Staubli VAL3: page.pgx

public program page(string& menuname[], num index)
// set all the page in english
begin
  //
  //  PAGE
  //
  //
  // PALLET PAGE
  if index>=10 and index<=19
    title("< Palettenseite >")
  endIf
  // PALLET VIEW PAGE
  if index>=100 and index<=109
    title("< Palettenanzeize >")
  endIf
  switch index
    //
    // PALLET
    //
    // Integrator programmer
    case 10,11
      menuname="Programm anzeigen,Edit Palette,,,Assistent,Reset,Zurück,Nächste"
    break
    // On Cycle
    case 13,14
      menuname="Programm anzeigen,Edit Palette,,,,Reset,Zurück,Nächste"
    break
    // VIEW PALLET
    case 100,101,102,103,104,105
      menuname="Reset ALLES,,,,,Reset,Zurück,Nächste"
    break
  endSwitch
end
